FUNCTION_BLOCK FB_AxisOP
VAR_INPUT
	bEnable: BOOL;
	stHardware: ST_AxisHardware;
END_VAR
VAR_OUTPUT
	bDone: BOOL;
	bBusy: BOOL;
	bError: BOOL;
	nErrorID: UDINT;
	currDriveState: ST_EcSlaveState;
	currEncState: ST_EcSlaveState;
END_VAR
VAR
	fbSetDriveState: FB_EcSetSlaveState;
	fbSetEncState: FB_EcSetSlaveState;
	bDriveDone: BOOL;
	bEncDone: BOOL;
	bDriveBusy: BOOL;
	bEncBusy: BOOL;
	bDriveErr: BOOL;
	bEncErr: BOOL;
	nDriveErrID: UDINT;
	nEncErrID: UDINT;
END_VAR

// Only do it once
IF bEnable AND NOT bDone THEN
	IF stHardware.drive_type = 0 THEN
		bDriveDone := TRUE;
		bDriveBusy := FALSE;
		bDriveErr := FALSE;
		nDriveErrID := 0;
	ELSE
		fbSetDriveState(sNetID:=stHardware.drive_ref.sNetId,
			nSlaveAddr:=stHardware.drive_ref.nSlaveAddr,
			bExecute:=bEnable,
			reqState:=EC_DEVICE_STATE_OP,
			bBusy=>bDriveBusy,
			bError=>bDriveErr,
			nErrId=>nDriveErrID,
			currState=>currDriveState);
		bDriveDone := bEnable AND NOT fbSetDriveState.bBusy AND currDriveState.deviceState = EC_DEVICE_STATE_OP;
	END_IF
	IF stHardware.enc_type = 0 THEN
		bEncDone := TRUE;
		bEncBusy := FALSE;
		bEncErr := FALSE;
		nEncErrID := 0;
	ELSE
		fbSetEncState(sNetID:=stHardware.enc_ref.sNetId,
			nSlaveAddr:=stHardware.enc_ref.nSlaveAddr,
			bExecute:=bEnable,
			reqState:=EC_DEVICE_STATE_OP,
			bBusy=>bEncBusy,
			bError=>bEncErr,
			nErrId=>nEncErrID,
			currState=>currEncState);
		bEncDone := bEnable AND NOT fbSetEncState.bBusy AND currEncState.deviceState = EC_DEVICE_STATE_OP;
	END_IF
END_IF
bDone := bDriveDone AND bEncDone;
bBusy := bDriveBusy OR bEncBusy;
bError := bDriveErr OR bEncErr;
IF nDriveErrID > 0 THEN
	nErrorID := nDriveErrID;
ELSE
	nErrorID := nEncErrID;
END_IF

END_FUNCTION_BLOCK

(* stored: Version 1.1.0.1, ProductVersion 3.1.4020.12
   POU FB_AxisOP: Id {2d312ae8-fcfa-4504-9380-5754eab57884}, SpecialFunc None *)
